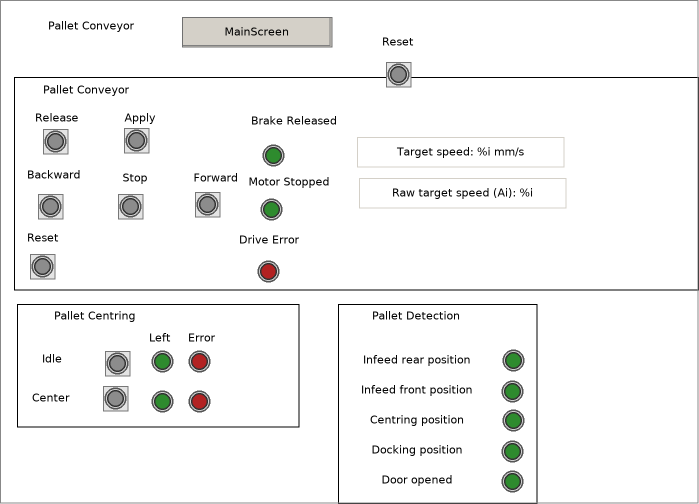
VISUALIZATION PalletConveyor  // 699x504
    Rectangle (14,77 685x213)
    Rectangle (17,304 282x123)
    Label (16,11 150x30), "Pallet Conveyor"
    Button (182,17 150x30), "MainScreen"
        OnMouseClick: change screen: MainScreen
    Lamp1 (261,143 25x25), variable: GVL_Modules.g_emPalletConveyor.s_cmPalletConveyor.s_fbHmiLedBrakeReleased.i_bStaLed, style: Lamp-Lamp1-Green
    Lamp1 (256,259 25x25), variable: GVL_Modules.g_emPalletConveyor.s_cmPalletConveyor.s_fbHmiLedDriveError.i_bStaLed, style: Lamp-Lamp1-Red
    Label (219,106 150x30), "Brake Released"
    Label (194,225 150x30), "Drive Error"
    Lamp1 (259,197 25x25), variable: GVL_Modules.g_emPalletConveyor.s_cmPalletConveyor.s_fbHmiLedMotorStopped.i_bStaLed, style: Lamp-Lamp1-Green
    Label (214,167 150x30), "Motor Stopped"
    PushSwitch (124,128 25x25), variable: GVL_Modules.g_emPalletConveyor.s_cmPalletConveyor.s_fbHmiBtnManualApplyBrake.s_bFromHmiPressed, behaviour: TAP, style: Switch-PushSwitch-Gray
    PushSwitch (43,129 25x25), variable: GVL_Modules.g_emPalletConveyor.s_cmPalletConveyor.s_fbHmiBtnManualReleaseBrake.s_bFromHmiPressed, behaviour: TAP, style: Switch-PushSwitch-Gray
    PushSwitch (38,194 25x25), variable: GVL_Modules.g_emPalletConveyor.s_cmPalletConveyor.s_fbHmiBtnManualBackward.s_bFromHmiPressed, behaviour: TAP, style: Switch-PushSwitch-Gray
    PushSwitch (118,194 25x25), variable: GVL_Modules.g_emPalletConveyor.s_cmPalletConveyor.s_fbHmiBtnManualStop.s_bFromHmiPressed, behaviour: TAP, style: Switch-PushSwitch-Gray
    PushSwitch (195,192 25x25), variable: GVL_Modules.g_emPalletConveyor.s_cmPalletConveyor.s_fbHmiBtnManualForward.s_bFromHmiPressed, behaviour: TAP, style: Switch-PushSwitch-Gray
    Label (18,103 78x30), "Release"
    Label (101,103 78x30), "Apply"
    Label (15,160 78x30), "Backward"
    Label (96,163 78x30), "Stop"
    Label (177,163 78x30), "Forward"
    PushSwitch (30,254 25x25), variable: GVL_Modules.g_emPalletConveyor.s_cmPalletConveyor.s_fbHmiBtnManualReset.s_bFromHmiPressed, behaviour: TAP, style: Switch-PushSwitch-Gray
    Label (4,223 78x30), "Reset"
    Textfield (359,178 207x30), "Raw target speed (Ai): %i", text variable: GVL_Modules.g_emPalletConveyor.s_cmPalletConveyor.Q_nSetTargetSpeed
    Textfield (357,137 207x30), "Target speed: %i mm/s", text variable: GVL_Modules.g_emPalletConveyor.s_cmPalletConveyor.s_rTargetSpeed, input disabled if: 0
        OnMouseClick: write the text variable via VisuDialogs.Numpad, min 40, max 200
    Label (11,75 150x30), "Pallet Conveyor"
    Lamp1 (150,349 25x25), variable: GVL_Modules.g_emPalletConveyor.s_cmCentringUnit.s_fbHmiLedIsOff.i_bStaLed, style: Lamp-Lamp1-Green
    Lamp1 (187,349 25x25), variable: GVL_Modules.g_emPalletConveyor.s_cmCentringUnit.s_fbHmiLedErrorOff.i_bStaLed, style: Lamp-Lamp1-Red
    Label (107,323 150x30), "Left Error"
    PushSwitch (103,386 25x25), variable: GVL_Modules.g_emPalletConveyor.s_cmCentringUnit.s_fbHmiBtnManualOn.s_bFromHmiPressed, behaviour: TAP, style: Switch-PushSwitch-Gray
    PushSwitch (105,351 25x25), variable: GVL_Modules.g_emPalletConveyor.s_cmCentringUnit.s_fbHmiBtnManualOff.s_bFromHmiPressed, behaviour: TAP, style: Switch-PushSwitch-Gray
    Label (13,344 78x30), "Idle"
    Label (12,383 78x30), "Center"
    Label (24,386 78x30)
    Label (186,389 78x30)
    Label (7,438 78x30)
    Label (20,301 150x30), "Pallet Centring"
    Lamp1 (150,389 25x25), variable: GVL_Modules.g_emPalletConveyor.s_cmCentringUnit.s_fbHmiLedIsOn.i_bStaLed, style: Lamp-Lamp1-Green
    Lamp1 (187,389 25x25), variable: GVL_Modules.g_emPalletConveyor.s_cmCentringUnit.s_fbHmiLedErrorOn.i_bStaLed, style: Lamp-Lamp1-Red
    PushSwitch (386,62 25x25), variable: GVL.g_unCleanroomConnect.s_fbHmiBtnReset.s_bFromHmiPressed, behaviour: TAP, style: Switch-PushSwitch-Gray
    Label (359,27 78x30), "Reset"
    Rectangle (338,304 199x200)
    Lamp1 (501,348 25x25), variable: GVL_Modules.g_emPalletConveyor.s_fbHmiLedInfeedRearPosition.i_bStaLed, style: Lamp-Lamp1-Green
    Label (348,345 138x30), "Infeed rear position"
    Label (345,386 78x30)
    Label (341,301 150x30), "Pallet Detection"
    Lamp1 (500,379 25x25), variable: GVL_Modules.g_emPalletConveyor.s_fbHmiLedInfeedFrontPosition.i_bStaLed, style: Lamp-Lamp1-Green
    Lamp1 (501,408 25x25), variable: GVL_Modules.g_emPalletConveyor.s_fbHmiLedCentringPosition.i_bStaLed, style: Lamp-Lamp1-Green
    Lamp1 (500,439 25x25), variable: GVL_Modules.g_emPalletConveyor.s_fbHmiLedDockingPosition.i_bStaLed, style: Lamp-Lamp1-Green
    Lamp1 (500,469 25x25), variable: GVL_Modules.g_emPalletConveyor.s_cmCentringUnit.s_fbHmiLedIsOn.i_bStaLed, style: Lamp-Lamp1-Green
    Label (348,375 138x30), "Infeed front position"
    Label (348,405 138x30), "Centring position"
    Label (348,435 138x30), "Docking position"
    Label (348,465 138x30), "Door opened"
END_VISUALIZATION

(* stored: Version 1.1.0.1, ProductVersion 3.1.4024.12
   Visu PalletConveyor: Id {2841a37d-bd22-4f18-9265-0c86f99f4b7e} *)
